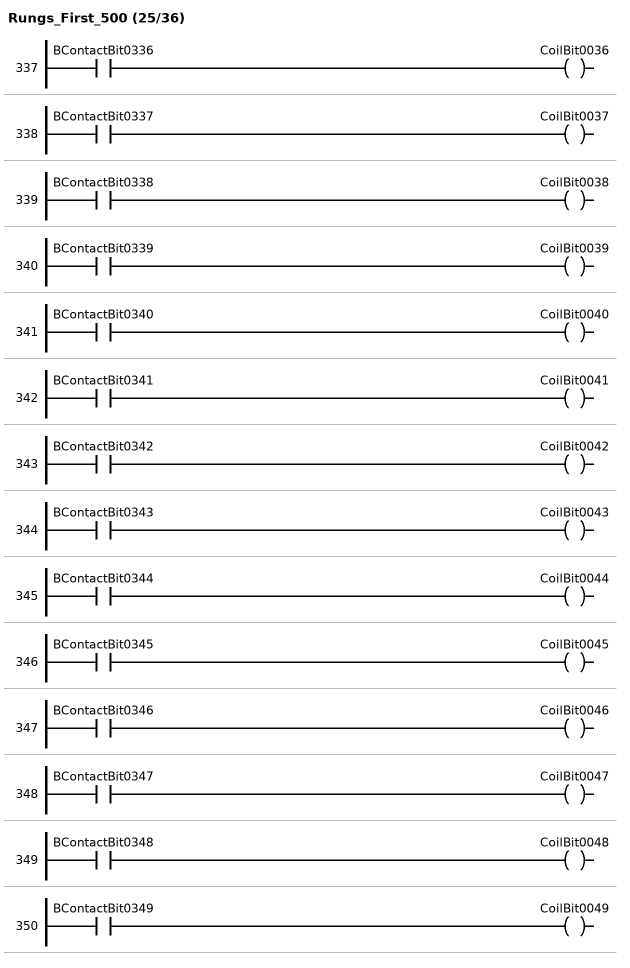
// NETWORK 337
CoilBit0036 := BContactBit0336;

// NETWORK 338
CoilBit0037 := BContactBit0337;

// NETWORK 339
CoilBit0038 := BContactBit0338;

// NETWORK 340
CoilBit0039 := BContactBit0339;

// NETWORK 341
CoilBit0040 := BContactBit0340;

// NETWORK 342
CoilBit0041 := BContactBit0341;

// NETWORK 343
CoilBit0042 := BContactBit0342;

// NETWORK 344
CoilBit0043 := BContactBit0343;

// NETWORK 345
CoilBit0044 := BContactBit0344;

// NETWORK 346
CoilBit0045 := BContactBit0345;

// NETWORK 347
CoilBit0046 := BContactBit0346;

// NETWORK 348
CoilBit0047 := BContactBit0347;

// NETWORK 349
CoilBit0048 := BContactBit0348;

// NETWORK 350
CoilBit0049 := BContactBit0349;

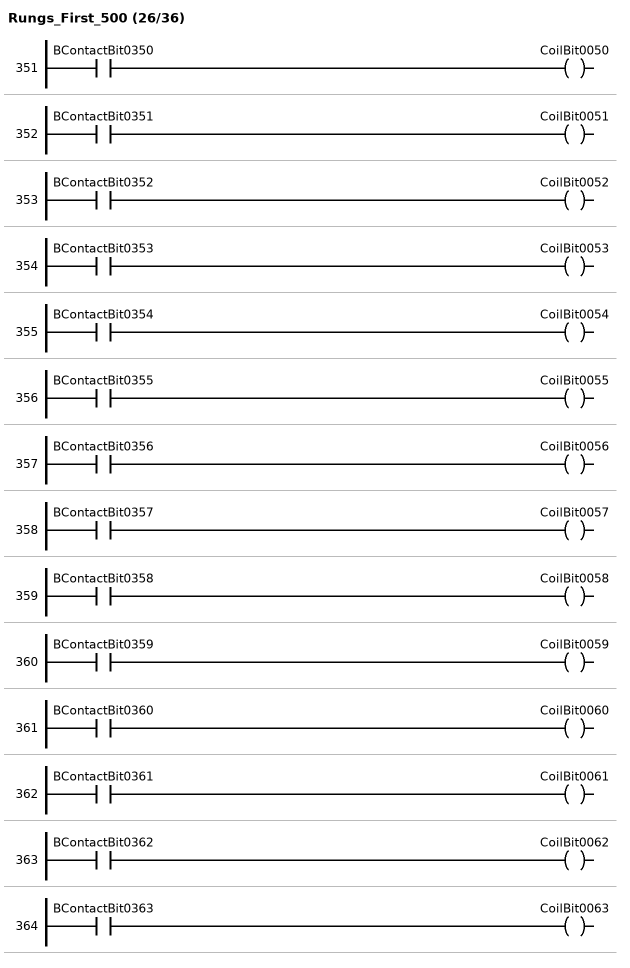
// NETWORK 351
CoilBit0050 := BContactBit0350;

// NETWORK 352
CoilBit0051 := BContactBit0351;

// NETWORK 353
CoilBit0052 := BContactBit0352;

// NETWORK 354
CoilBit0053 := BContactBit0353;

// NETWORK 355
CoilBit0054 := BContactBit0354;

// NETWORK 356
CoilBit0055 := BContactBit0355;

// NETWORK 357
CoilBit0056 := BContactBit0356;

// NETWORK 358
CoilBit0057 := BContactBit0357;

// NETWORK 359
CoilBit0058 := BContactBit0358;

// NETWORK 360
CoilBit0059 := BContactBit0359;

// NETWORK 361
CoilBit0060 := BContactBit0360;

// NETWORK 362
CoilBit0061 := BContactBit0361;

// NETWORK 363
CoilBit0062 := BContactBit0362;

// NETWORK 364
CoilBit0063 := BContactBit0363;

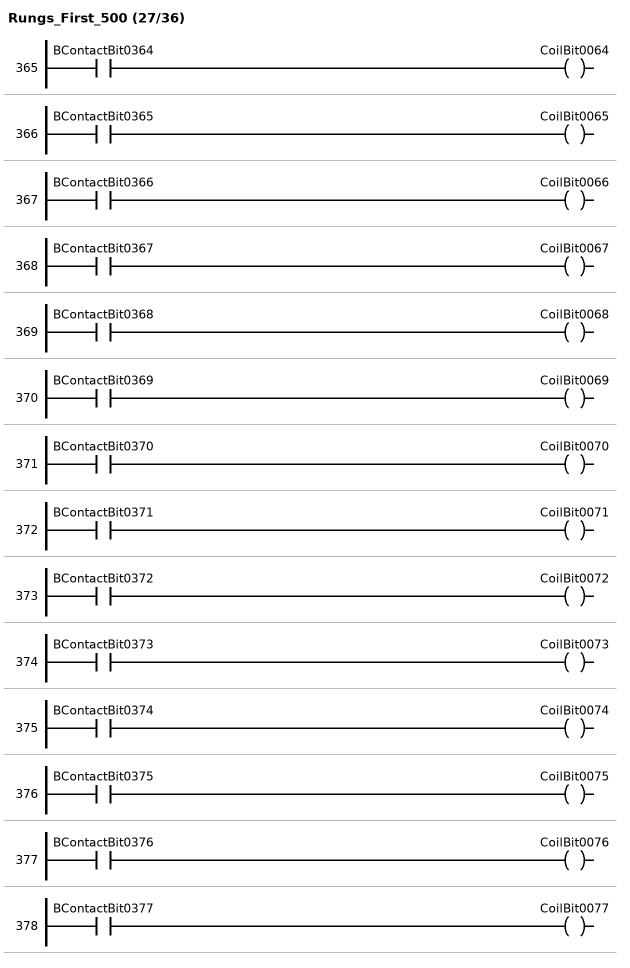
// NETWORK 365
CoilBit0064 := BContactBit0364;

// NETWORK 366
CoilBit0065 := BContactBit0365;

// NETWORK 367
CoilBit0066 := BContactBit0366;

// NETWORK 368
CoilBit0067 := BContactBit0367;

// NETWORK 369
CoilBit0068 := BContactBit0368;

// NETWORK 370
CoilBit0069 := BContactBit0369;

// NETWORK 371
CoilBit0070 := BContactBit0370;

// NETWORK 372
CoilBit0071 := BContactBit0371;

// NETWORK 373
CoilBit0072 := BContactBit0372;

// NETWORK 374
CoilBit0073 := BContactBit0373;

// NETWORK 375
CoilBit0074 := BContactBit0374;

// NETWORK 376
CoilBit0075 := BContactBit0375;

// NETWORK 377
CoilBit0076 := BContactBit0376;

// NETWORK 378
CoilBit0077 := BContactBit0377;

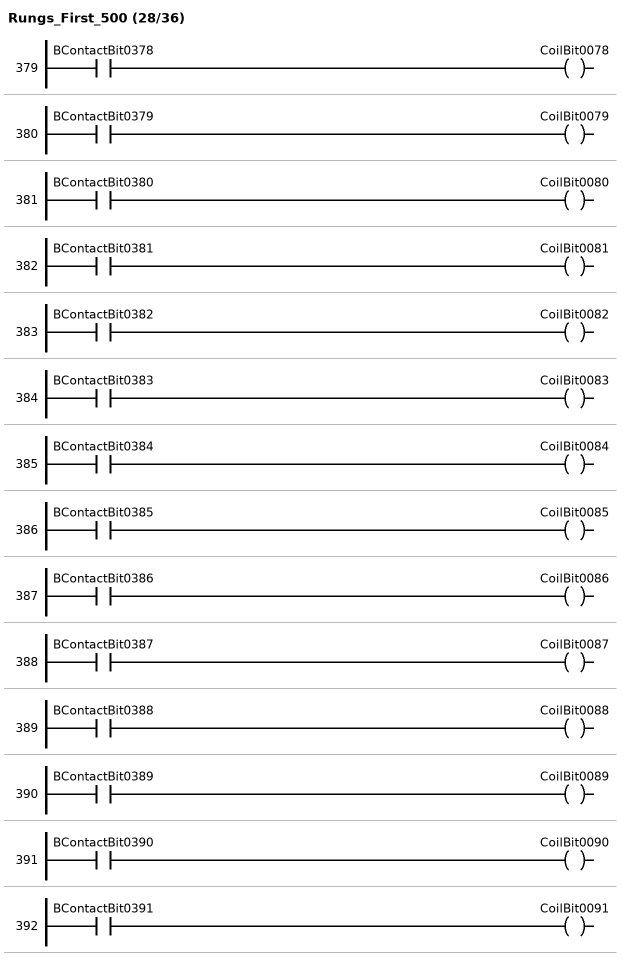
// NETWORK 379
CoilBit0078 := BContactBit0378;

// NETWORK 380
CoilBit0079 := BContactBit0379;

// NETWORK 381
CoilBit0080 := BContactBit0380;

// NETWORK 382
CoilBit0081 := BContactBit0381;

// NETWORK 383
CoilBit0082 := BContactBit0382;

// NETWORK 384
CoilBit0083 := BContactBit0383;

// NETWORK 385
CoilBit0084 := BContactBit0384;

// NETWORK 386
CoilBit0085 := BContactBit0385;

// NETWORK 387
CoilBit0086 := BContactBit0386;

// NETWORK 388
CoilBit0087 := BContactBit0387;

// NETWORK 389
CoilBit0088 := BContactBit0388;

// NETWORK 390
CoilBit0089 := BContactBit0389;

// NETWORK 391
CoilBit0090 := BContactBit0390;

// NETWORK 392
CoilBit0091 := BContactBit0391;

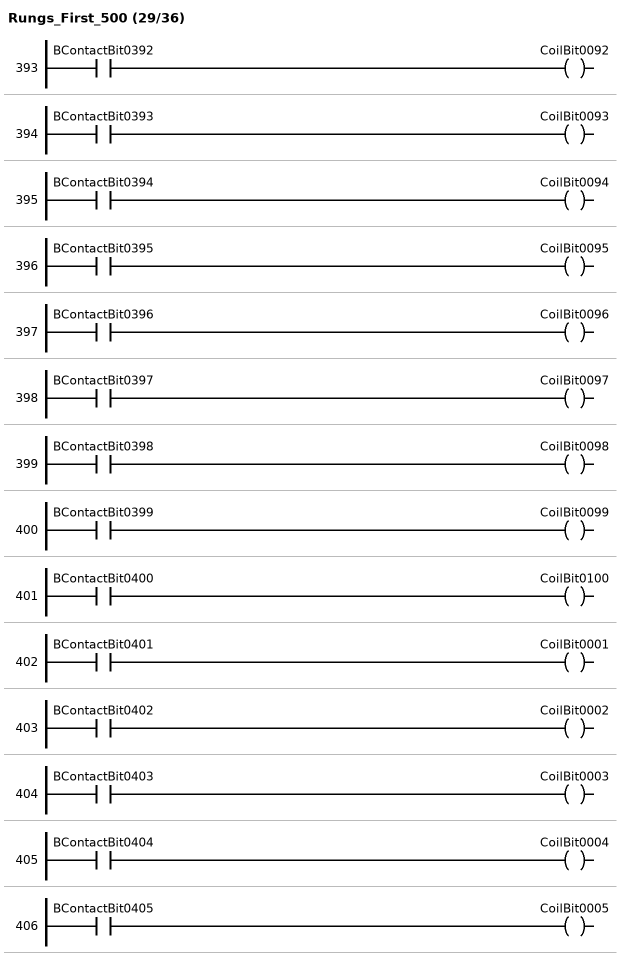
// NETWORK 393
CoilBit0092 := BContactBit0392;

// NETWORK 394
CoilBit0093 := BContactBit0393;

// NETWORK 395
CoilBit0094 := BContactBit0394;

// NETWORK 396
CoilBit0095 := BContactBit0395;

// NETWORK 397
CoilBit0096 := BContactBit0396;

// NETWORK 398
CoilBit0097 := BContactBit0397;

// NETWORK 399
CoilBit0098 := BContactBit0398;

// NETWORK 400
CoilBit0099 := BContactBit0399;

// NETWORK 401
CoilBit0100 := BContactBit0400;

// NETWORK 402
CoilBit0001 := BContactBit0401;

// NETWORK 403
CoilBit0002 := BContactBit0402;

// NETWORK 404
CoilBit0003 := BContactBit0403;

// NETWORK 405
CoilBit0004 := BContactBit0404;

// NETWORK 406
CoilBit0005 := BContactBit0405;

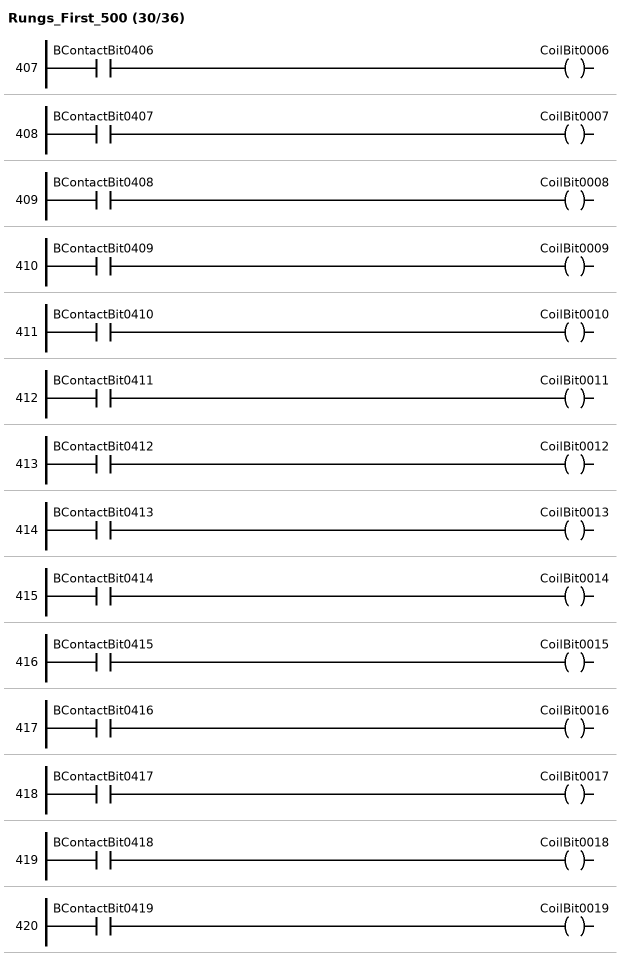
// NETWORK 407
CoilBit0006 := BContactBit0406;

// NETWORK 408
CoilBit0007 := BContactBit0407;

// NETWORK 409
CoilBit0008 := BContactBit0408;

// NETWORK 410
CoilBit0009 := BContactBit0409;

// NETWORK 411
CoilBit0010 := BContactBit0410;

// NETWORK 412
CoilBit0011 := BContactBit0411;

// NETWORK 413
CoilBit0012 := BContactBit0412;

// NETWORK 414
CoilBit0013 := BContactBit0413;

// NETWORK 415
CoilBit0014 := BContactBit0414;

// NETWORK 416
CoilBit0015 := BContactBit0415;

// NETWORK 417
CoilBit0016 := BContactBit0416;

// NETWORK 418
CoilBit0017 := BContactBit0417;

// NETWORK 419
CoilBit0018 := BContactBit0418;

// NETWORK 420
CoilBit0019 := BContactBit0419;

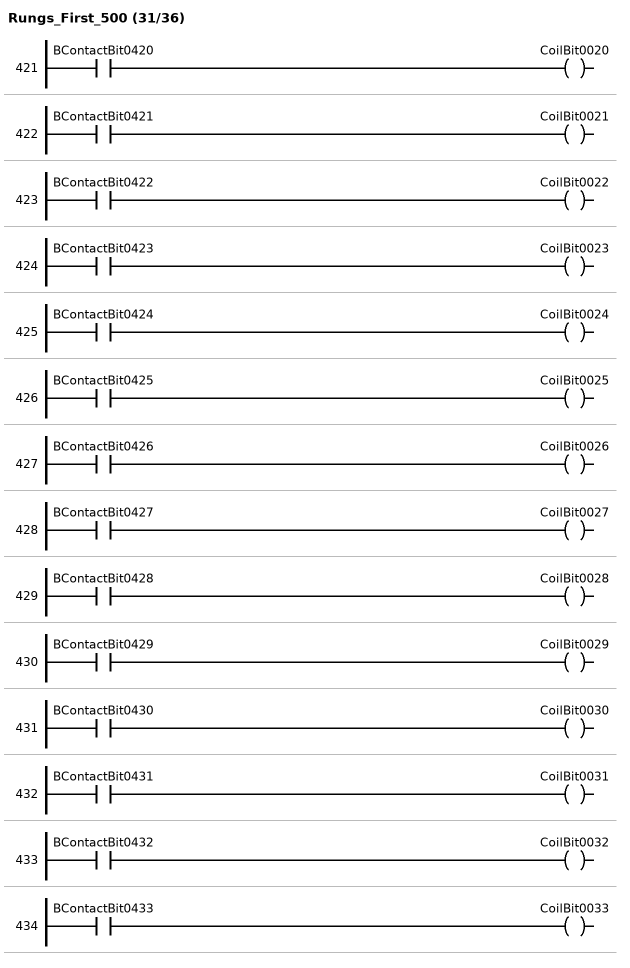
// NETWORK 421
CoilBit0020 := BContactBit0420;

// NETWORK 422
CoilBit0021 := BContactBit0421;

// NETWORK 423
CoilBit0022 := BContactBit0422;

// NETWORK 424
CoilBit0023 := BContactBit0423;

// NETWORK 425
CoilBit0024 := BContactBit0424;

// NETWORK 426
CoilBit0025 := BContactBit0425;

// NETWORK 427
CoilBit0026 := BContactBit0426;

// NETWORK 428
CoilBit0027 := BContactBit0427;

// NETWORK 429
CoilBit0028 := BContactBit0428;

// NETWORK 430
CoilBit0029 := BContactBit0429;

// NETWORK 431
CoilBit0030 := BContactBit0430;

// NETWORK 432
CoilBit0031 := BContactBit0431;

// NETWORK 433
CoilBit0032 := BContactBit0432;

// NETWORK 434
CoilBit0033 := BContactBit0433;

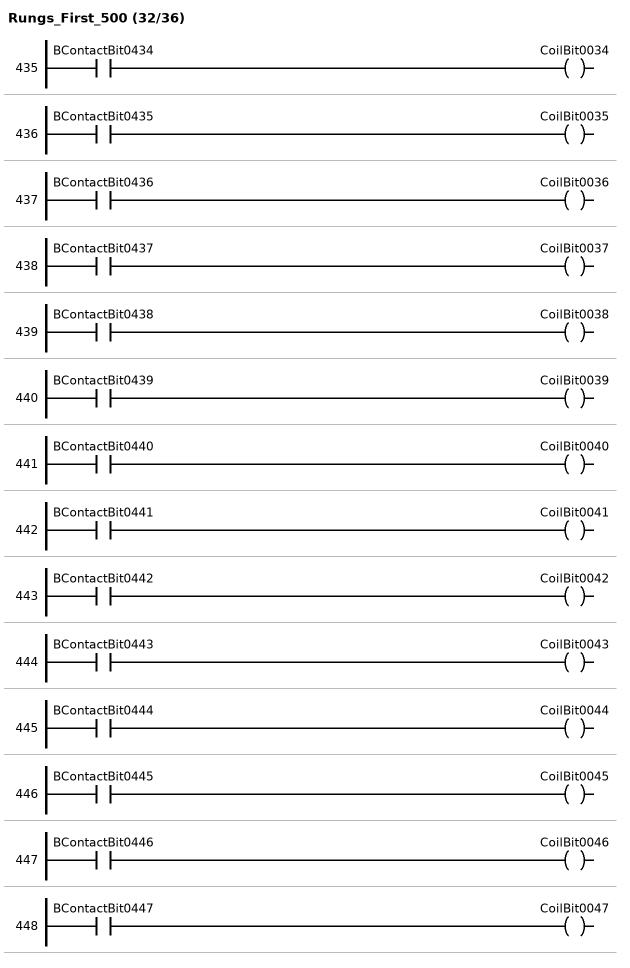
// NETWORK 435
CoilBit0034 := BContactBit0434;

// NETWORK 436
CoilBit0035 := BContactBit0435;

// NETWORK 437
CoilBit0036 := BContactBit0436;

// NETWORK 438
CoilBit0037 := BContactBit0437;

// NETWORK 439
CoilBit0038 := BContactBit0438;

// NETWORK 440
CoilBit0039 := BContactBit0439;

// NETWORK 441
CoilBit0040 := BContactBit0440;

// NETWORK 442
CoilBit0041 := BContactBit0441;

// NETWORK 443
CoilBit0042 := BContactBit0442;

// NETWORK 444
CoilBit0043 := BContactBit0443;

// NETWORK 445
CoilBit0044 := BContactBit0444;

// NETWORK 446
CoilBit0045 := BContactBit0445;

// NETWORK 447
CoilBit0046 := BContactBit0446;

// NETWORK 448
CoilBit0047 := BContactBit0447;

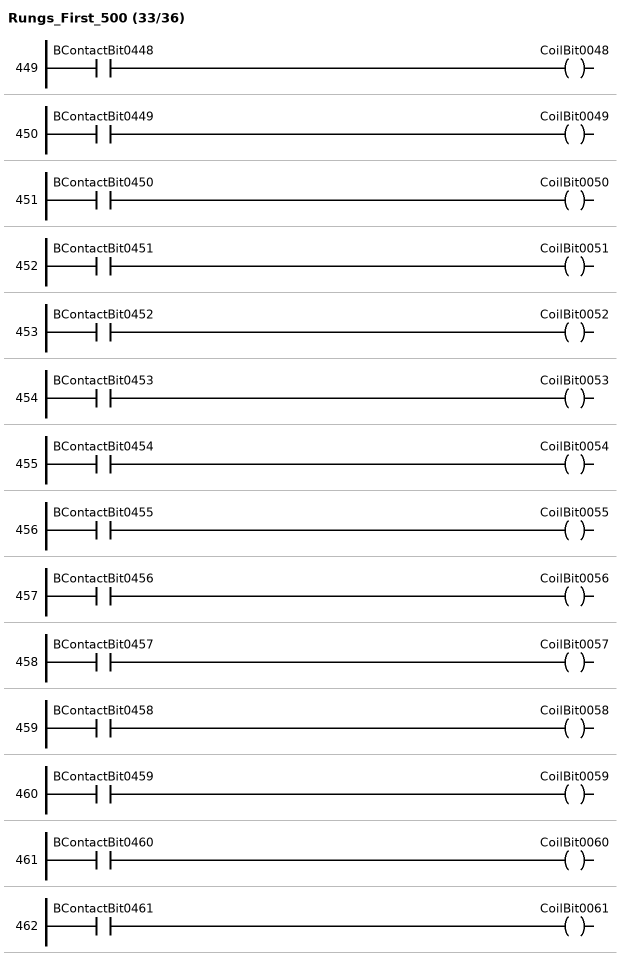
// NETWORK 449
CoilBit0048 := BContactBit0448;

// NETWORK 450
CoilBit0049 := BContactBit0449;

// NETWORK 451
CoilBit0050 := BContactBit0450;

// NETWORK 452
CoilBit0051 := BContactBit0451;

// NETWORK 453
CoilBit0052 := BContactBit0452;

// NETWORK 454
CoilBit0053 := BContactBit0453;

// NETWORK 455
CoilBit0054 := BContactBit0454;

// NETWORK 456
CoilBit0055 := BContactBit0455;

// NETWORK 457
CoilBit0056 := BContactBit0456;

// NETWORK 458
CoilBit0057 := BContactBit0457;

// NETWORK 459
CoilBit0058 := BContactBit0458;

// NETWORK 460
CoilBit0059 := BContactBit0459;

// NETWORK 461
CoilBit0060 := BContactBit0460;

// NETWORK 462
CoilBit0061 := BContactBit0461;

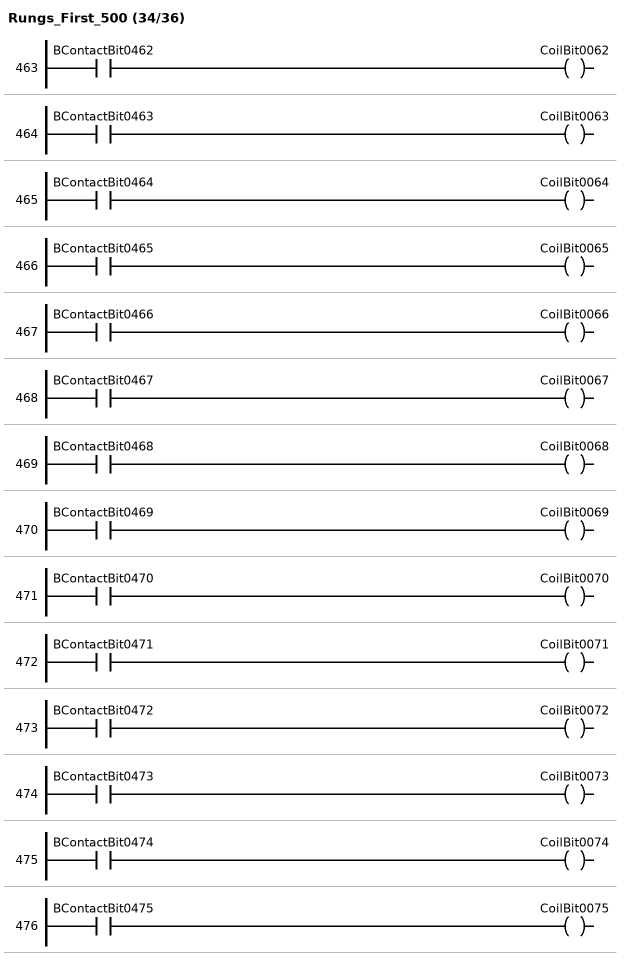
// NETWORK 463
CoilBit0062 := BContactBit0462;

// NETWORK 464
CoilBit0063 := BContactBit0463;

// NETWORK 465
CoilBit0064 := BContactBit0464;

// NETWORK 466
CoilBit0065 := BContactBit0465;

// NETWORK 467
CoilBit0066 := BContactBit0466;

// NETWORK 468
CoilBit0067 := BContactBit0467;

// NETWORK 469
CoilBit0068 := BContactBit0468;

// NETWORK 470
CoilBit0069 := BContactBit0469;

// NETWORK 471
CoilBit0070 := BContactBit0470;

// NETWORK 472
CoilBit0071 := BContactBit0471;

// NETWORK 473
CoilBit0072 := BContactBit0472;

// NETWORK 474
CoilBit0073 := BContactBit0473;

// NETWORK 475
CoilBit0074 := BContactBit0474;

// NETWORK 476
CoilBit0075 := BContactBit0475;

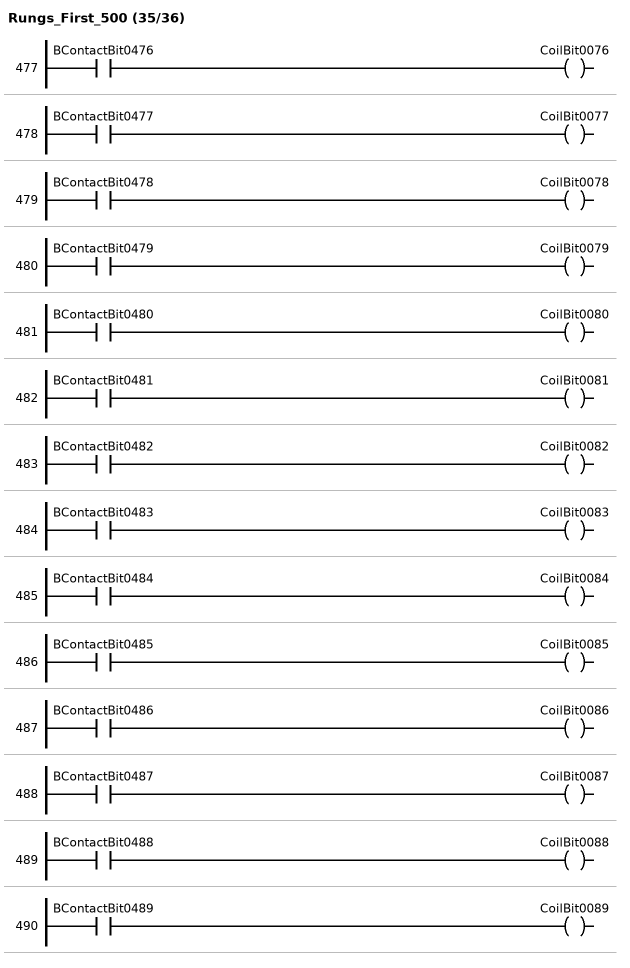
// NETWORK 477
CoilBit0076 := BContactBit0476;

// NETWORK 478
CoilBit0077 := BContactBit0477;

// NETWORK 479
CoilBit0078 := BContactBit0478;

// NETWORK 480
CoilBit0079 := BContactBit0479;

// NETWORK 481
CoilBit0080 := BContactBit0480;

// NETWORK 482
CoilBit0081 := BContactBit0481;

// NETWORK 483
CoilBit0082 := BContactBit0482;

// NETWORK 484
CoilBit0083 := BContactBit0483;

// NETWORK 485
CoilBit0084 := BContactBit0484;

// NETWORK 486
CoilBit0085 := BContactBit0485;

// NETWORK 487
CoilBit0086 := BContactBit0486;

// NETWORK 488
CoilBit0087 := BContactBit0487;

// NETWORK 489
CoilBit0088 := BContactBit0488;

// NETWORK 490
CoilBit0089 := BContactBit0489;

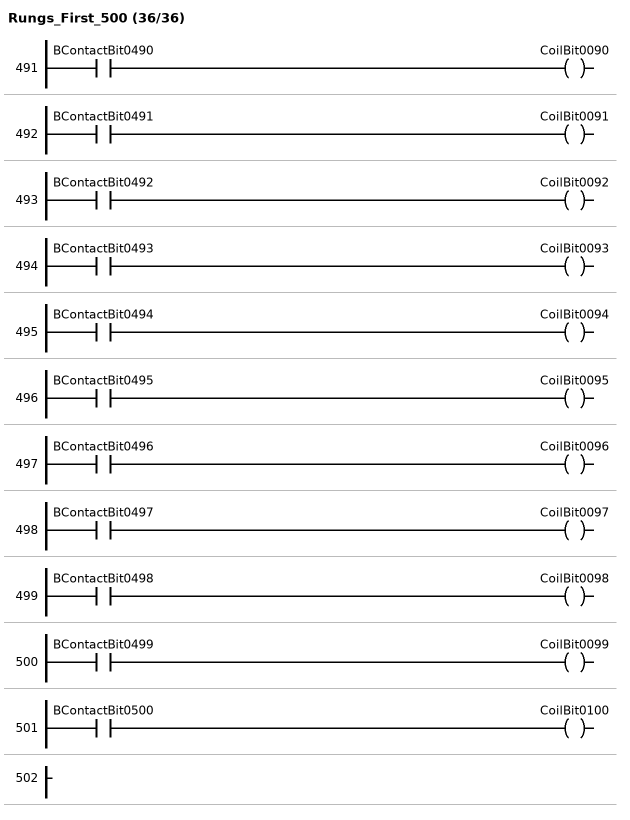
// NETWORK 491
CoilBit0090 := BContactBit0490;

// NETWORK 492
CoilBit0091 := BContactBit0491;

// NETWORK 493
CoilBit0092 := BContactBit0492;

// NETWORK 494
CoilBit0093 := BContactBit0493;

// NETWORK 495
CoilBit0094 := BContactBit0494;

// NETWORK 496
CoilBit0095 := BContactBit0495;

// NETWORK 497
CoilBit0096 := BContactBit0496;

// NETWORK 498
CoilBit0097 := BContactBit0497;

// NETWORK 499
CoilBit0098 := BContactBit0498;

// NETWORK 500
CoilBit0099 := BContactBit0499;

// NETWORK 501
CoilBit0100 := BContactBit0500;

// NETWORK 502

END_PROGRAM

// Rungs_Second_500
PROGRAM Rungs_Second_500
VAR

ContactBit0000	:BOOL;
ContactBit0001	:BOOL;
ContactBit0002	:BOOL;
ContactBit0003	:BOOL;
ContactBit0004	:BOOL;
ContactBit0005	:BOOL;
ContactBit0006	:BOOL;
ContactBit0007	:BOOL;
ContactBit0008	:BOOL;
ContactBit0009	:BOOL;
ContactBit0010	:BOOL;
ContactBit0011	:BOOL;
ContactBit0012	:BOOL;
ContactBit0013	:BOOL;
ContactBit0014	:BOOL;
ContactBit0015	:BOOL;
ContactBit0016	:BOOL;
ContactBit0017	:BOOL;
ContactBit0018	:BOOL;
ContactBit0019	:BOOL;
ContactBit0020	:BOOL;
ContactBit0021	:BOOL;
ContactBit0022	:BOOL;
ContactBit0023	:BOOL;
ContactBit0024	:BOOL;
ContactBit0025	:BOOL;
ContactBit0026	:BOOL;
ContactBit0027	:BOOL;
ContactBit0028	:BOOL;
ContactBit0029	:BOOL;
ContactBit0030	:BOOL;
ContactBit0031	:BOOL;
ContactBit0032	:BOOL;
ContactBit0033	:BOOL;
ContactBit0034	:BOOL;
ContactBit0035	:BOOL;
ContactBit0036	:BOOL;
ContactBit0037	:BOOL;
ContactBit0038	:BOOL;
ContactBit0039	:BOOL;
ContactBit0040	:BOOL;
ContactBit0041	:BOOL;
ContactBit0042	:BOOL;
ContactBit0043	:BOOL;
ContactBit0044	:BOOL;
ContactBit0045	:BOOL;
ContactBit0046	:BOOL;
ContactBit0047	:BOOL;
ContactBit0048	:BOOL;
ContactBit0049	:BOOL;
ContactBit0050	:BOOL;
ContactBit0051	:BOOL;
ContactBit0052	:BOOL;
ContactBit0053	:BOOL;
ContactBit0054	:BOOL;
ContactBit0055	:BOOL;
ContactBit0056	:BOOL;
ContactBit0057	:BOOL;
ContactBit0058	:BOOL;
ContactBit0059	:BOOL;
ContactBit0060	:BOOL;
ContactBit0061	:BOOL;
ContactBit0062	:BOOL;
ContactBit0063	:BOOL;
ContactBit0064	:BOOL;
ContactBit0065	:BOOL;
ContactBit0066	:BOOL;
ContactBit0067	:BOOL;
ContactBit0068	:BOOL;
ContactBit0069	:BOOL;
ContactBit0070	:BOOL;
ContactBit0071	:BOOL;
ContactBit0072	:BOOL;
ContactBit0073	:BOOL;
ContactBit0074	:BOOL;
ContactBit0075	:BOOL;
ContactBit0076	:BOOL;
ContactBit0077	:BOOL;
ContactBit0078	:BOOL;
ContactBit0079	:BOOL;
ContactBit0080	:BOOL;
ContactBit0081	:BOOL;
ContactBit0082	:BOOL;
ContactBit0083	:BOOL;
ContactBit0084	:BOOL;
ContactBit0085	:BOOL;
ContactBit0086	:BOOL;
ContactBit0087	:BOOL;
ContactBit0088	:BOOL;
ContactBit0089	:BOOL;
ContactBit0090	:BOOL;
ContactBit0091	:BOOL;
ContactBit0092	:BOOL;
ContactBit0093	:BOOL;
ContactBit0094	:BOOL;
ContactBit0095	:BOOL;
ContactBit0096	:BOOL;
ContactBit0097	:BOOL;
ContactBit0098	:BOOL;
ContactBit0099	:BOOL;
ContactBit0100	:BOOL;
ContactBit0101	:BOOL;
ContactBit0102	:BOOL;
ContactBit0103	:BOOL;
ContactBit0104	:BOOL;
ContactBit0105	:BOOL;
ContactBit0106	:BOOL;
ContactBit0107	:BOOL;
ContactBit0108	:BOOL;
ContactBit0109	:BOOL;
ContactBit0110	:BOOL;
ContactBit0111	:BOOL;
ContactBit0112	:BOOL;
ContactBit0113	:BOOL;
ContactBit0114	:BOOL;
ContactBit0115	:BOOL;
ContactBit0116	:BOOL;
ContactBit0117	:BOOL;
ContactBit0118	:BOOL;
ContactBit0119	:BOOL;
ContactBit0120	:BOOL;
ContactBit0121	:BOOL;
ContactBit0122	:BOOL;
ContactBit0123	:BOOL;
ContactBit0124	:BOOL;
ContactBit0125	:BOOL;
ContactBit0126	:BOOL;
ContactBit0127	:BOOL;
ContactBit0128	:BOOL;
ContactBit0129	:BOOL;
ContactBit0130	:BOOL;
ContactBit0131	:BOOL;
ContactBit0132	:BOOL;
ContactBit0133	:BOOL;
ContactBit0134	:BOOL;
ContactBit0135	:BOOL;
ContactBit0136	:BOOL;
ContactBit0137	:BOOL;
ContactBit0138	:BOOL;
ContactBit0139	:BOOL;
ContactBit0140	:BOOL;
ContactBit0141	:BOOL;
ContactBit0142	:BOOL;
ContactBit0143	:BOOL;
ContactBit0144	:BOOL;
ContactBit0145	:BOOL;
ContactBit0146	:BOOL;
ContactBit0147	:BOOL;
ContactBit0148	:BOOL;
ContactBit0149	:BOOL;
ContactBit0150	:BOOL;
ContactBit0151	:BOOL;
ContactBit0152	:BOOL;
ContactBit0153	:BOOL;
ContactBit0154	:BOOL;
ContactBit0155	:BOOL;
ContactBit0156	:BOOL;
ContactBit0157	:BOOL;
ContactBit0158	:BOOL;
ContactBit0159	:BOOL;
ContactBit0160	:BOOL;
ContactBit0161	:BOOL;
ContactBit0162	:BOOL;
ContactBit0163	:BOOL;
ContactBit0164	:BOOL;
ContactBit0165	:BOOL;
ContactBit0166	:BOOL;
ContactBit0167	:BOOL;
ContactBit0168	:BOOL;
ContactBit0169	:BOOL;
ContactBit0170	:BOOL;
ContactBit0171	:BOOL;
ContactBit0172	:BOOL;
ContactBit0173	:BOOL;
ContactBit0174	:BOOL;
ContactBit0175	:BOOL;
ContactBit0176	:BOOL;
ContactBit0177	:BOOL;
ContactBit0178	:BOOL;
ContactBit0179	:BOOL;
ContactBit0180	:BOOL;
ContactBit0181	:BOOL;
ContactBit0182	:BOOL;
ContactBit0183	:BOOL;
ContactBit0184	:BOOL;
ContactBit0185	:BOOL;
ContactBit0186	:BOOL;
ContactBit0187	:BOOL;
ContactBit0188	:BOOL;
ContactBit0189	:BOOL;
ContactBit0190	:BOOL;
ContactBit0191	:BOOL;
ContactBit0192	:BOOL;
ContactBit0193	:BOOL;
ContactBit0194	:BOOL;
ContactBit0195	:BOOL;
ContactBit0196	:BOOL;
ContactBit0197	:BOOL;
ContactBit0198	:BOOL;
ContactBit0199	:BOOL;
ContactBit0200	:BOOL;
ContactBit0201	:BOOL;
ContactBit0202	:BOOL;
ContactBit0203	:BOOL;
ContactBit0204	:BOOL;
ContactBit0205	:BOOL;
ContactBit0206	:BOOL;
ContactBit0207	:BOOL;
ContactBit0208	:BOOL;
ContactBit0209	:BOOL;
ContactBit0210	:BOOL;
ContactBit0211	:BOOL;
ContactBit0212	:BOOL;
ContactBit0213	:BOOL;
ContactBit0214	:BOOL;
ContactBit0215	:BOOL;
ContactBit0216	:BOOL;
ContactBit0217	:BOOL;
ContactBit0218	:BOOL;
ContactBit0219	:BOOL;
ContactBit0220	:BOOL;
ContactBit0221	:BOOL;
ContactBit0222	:BOOL;
ContactBit0223	:BOOL;
ContactBit0224	:BOOL;
ContactBit0225	:BOOL;
ContactBit0226	:BOOL;
ContactBit0227	:BOOL;
ContactBit0228	:BOOL;
ContactBit0229	:BOOL;
ContactBit0230	:BOOL;
ContactBit0231	:BOOL;
ContactBit0232	:BOOL;
ContactBit0233	:BOOL;
ContactBit0234	:BOOL;
ContactBit0235	:BOOL;
ContactBit0236	:BOOL;
ContactBit0237	:BOOL;
ContactBit0238	:BOOL;
ContactBit0239	:BOOL;
ContactBit0240	:BOOL;
ContactBit0241	:BOOL;
ContactBit0242	:BOOL;
ContactBit0243	:BOOL;
ContactBit0244	:BOOL;
ContactBit0245	:BOOL;
ContactBit0246	:BOOL;
ContactBit0247	:BOOL;
ContactBit0248	:BOOL;
ContactBit0249	:BOOL;
ContactBit0250	:BOOL;
ContactBit0251	:BOOL;
ContactBit0252	:BOOL;
ContactBit0253	:BOOL;
ContactBit0254	:BOOL;
ContactBit0255	:BOOL;
ContactBit0256	:BOOL;
ContactBit0257	:BOOL;
ContactBit0258	:BOOL;
ContactBit0259	:BOOL;
ContactBit0260	:BOOL;
ContactBit0261	:BOOL;
ContactBit0262	:BOOL;
ContactBit0263	:BOOL;
ContactBit0264	:BOOL;
ContactBit0265	:BOOL;
ContactBit0266	:BOOL;
ContactBit0267	:BOOL;
ContactBit0268	:BOOL;
ContactBit0269	:BOOL;
ContactBit0270	:BOOL;
ContactBit0271	:BOOL;
ContactBit0272	:BOOL;
ContactBit0273	:BOOL;
ContactBit0274	:BOOL;
ContactBit0275	:BOOL;
ContactBit0276	:BOOL;
ContactBit0277	:BOOL;
ContactBit0278	:BOOL;
ContactBit0279	:BOOL;
ContactBit0280	:BOOL;
ContactBit0281	:BOOL;
ContactBit0282	:BOOL;
ContactBit0283	:BOOL;
ContactBit0284	:BOOL;
ContactBit0285	:BOOL;
ContactBit0286	:BOOL;
ContactBit0287	:BOOL;
ContactBit0288	:BOOL;
ContactBit0289	:BOOL;
ContactBit0290	:BOOL;
ContactBit0291	:BOOL;
ContactBit0292	:BOOL;
ContactBit0293	:BOOL;
ContactBit0294	:BOOL;
ContactBit0295	:BOOL;
ContactBit0296	:BOOL;
ContactBit0297	:BOOL;
ContactBit0298	:BOOL;
ContactBit0299	:BOOL;
ContactBit0300	:BOOL;
ContactBit0301	:BOOL;
ContactBit0302	:BOOL;
ContactBit0303	:BOOL;
ContactBit0304	:BOOL;
ContactBit0305	:BOOL;
ContactBit0306	:BOOL;
ContactBit0307	:BOOL;
ContactBit0308	:BOOL;
ContactBit0309	:BOOL;
ContactBit0310	:BOOL;
ContactBit0311	:BOOL;
ContactBit0312	:BOOL;
ContactBit0313	:BOOL;
ContactBit0314	:BOOL;
ContactBit0315	:BOOL;
ContactBit0316	:BOOL;
ContactBit0317	:BOOL;
ContactBit0318	:BOOL;
ContactBit0319	:BOOL;
ContactBit0320	:BOOL;
ContactBit0321	:BOOL;
ContactBit0322	:BOOL;
ContactBit0323	:BOOL;
ContactBit0324	:BOOL;
ContactBit0325	:BOOL;
ContactBit0326	:BOOL;
ContactBit0327	:BOOL;
ContactBit0328	:BOOL;
ContactBit0329	:BOOL;
ContactBit0330	:BOOL;
ContactBit0331	:BOOL;
ContactBit0332	:BOOL;
ContactBit0333	:BOOL;
ContactBit0334	:BOOL;
ContactBit0335	:BOOL;
ContactBit0336	:BOOL;
ContactBit0337	:BOOL;
ContactBit0338	:BOOL;
ContactBit0339	:BOOL;
ContactBit0340	:BOOL;
ContactBit0341	:BOOL;
ContactBit0342	:BOOL;
ContactBit0343	:BOOL;
ContactBit0344	:BOOL;
ContactBit0345	:BOOL;
ContactBit0346	:BOOL;
ContactBit0347	:BOOL;
ContactBit0348	:BOOL;
ContactBit0349	:BOOL;
ContactBit0350	:BOOL;
ContactBit0351	:BOOL;
ContactBit0352	:BOOL;
ContactBit0353	:BOOL;
ContactBit0354	:BOOL;
ContactBit0355	:BOOL;
ContactBit0356	:BOOL;
ContactBit0357	:BOOL;
ContactBit0358	:BOOL;
ContactBit0359	:BOOL;
ContactBit0360	:BOOL;
ContactBit0361	:BOOL;
ContactBit0362	:BOOL;
ContactBit0363	:BOOL;
ContactBit0364	:BOOL;
ContactBit0365	:BOOL;
ContactBit0366	:BOOL;
ContactBit0367	:BOOL;
ContactBit0368	:BOOL;
ContactBit0369	:BOOL;
ContactBit0370	:BOOL;
ContactBit0371	:BOOL;
ContactBit0372	:BOOL;
ContactBit0373	:BOOL;
ContactBit0374	:BOOL;
ContactBit0375	:BOOL;
ContactBit0376	:BOOL;
ContactBit0377	:BOOL;
ContactBit0378	:BOOL;
ContactBit0379	:BOOL;
ContactBit0380	:BOOL;
ContactBit0381	:BOOL;
ContactBit0382	:BOOL;
ContactBit0383	:BOOL;
ContactBit0384	:BOOL;
ContactBit0385	:BOOL;
ContactBit0386	:BOOL;
ContactBit0387	:BOOL;
ContactBit0388	:BOOL;
ContactBit0389	:BOOL;
ContactBit0390	:BOOL;
ContactBit0391	:BOOL;
ContactBit0392	:BOOL;
ContactBit0393	:BOOL;
ContactBit0394	:BOOL;
ContactBit0395	:BOOL;
ContactBit0396	:BOOL;
ContactBit0397	:BOOL;
ContactBit0398	:BOOL;
ContactBit0399	:BOOL;
ContactBit0400	:BOOL;
ContactBit0401	:BOOL;
ContactBit0402	:BOOL;
ContactBit0403	:BOOL;
ContactBit0404	:BOOL;
ContactBit0405	:BOOL;
ContactBit0406	:BOOL;
ContactBit0407	:BOOL;
ContactBit0408	:BOOL;
ContactBit0409	:BOOL;
ContactBit0410	:BOOL;
ContactBit0411	:BOOL;
ContactBit0412	:BOOL;
ContactBit0413	:BOOL;
ContactBit0414	:BOOL;
ContactBit0415	:BOOL;
ContactBit0416	:BOOL;
ContactBit0417	:BOOL;
ContactBit0418	:BOOL;
ContactBit0419	:BOOL;
ContactBit0420	:BOOL;
ContactBit0421	:BOOL;
ContactBit0422	:BOOL;
ContactBit0423	:BOOL;
ContactBit0424	:BOOL;
ContactBit0425	:BOOL;
ContactBit0426	:BOOL;
ContactBit0427	:BOOL;
ContactBit0428	:BOOL;
ContactBit0429	:BOOL;
ContactBit0430	:BOOL;
ContactBit0431	:BOOL;
ContactBit0432	:BOOL;
ContactBit0433	:BOOL;
ContactBit0434	:BOOL;
ContactBit0435	:BOOL;
ContactBit0436	:BOOL;
ContactBit0437	:BOOL;
ContactBit0438	:BOOL;
ContactBit0439	:BOOL;
ContactBit0440	:BOOL;
ContactBit0441	:BOOL;
ContactBit0442	:BOOL;
ContactBit0443	:BOOL;
ContactBit0444	:BOOL;
ContactBit0445	:BOOL;
ContactBit0446	:BOOL;
ContactBit0447	:BOOL;
ContactBit0448	:BOOL;
ContactBit0449	:BOOL;
ContactBit0450	:BOOL;
ContactBit0451	:BOOL;
ContactBit0452	:BOOL;
ContactBit0453	:BOOL;
ContactBit0454	:BOOL;
ContactBit0455	:BOOL;
ContactBit0456	:BOOL;
ContactBit0457	:BOOL;
ContactBit0458	:BOOL;
ContactBit0459	:BOOL;
ContactBit0460	:BOOL;
ContactBit0461	:BOOL;
ContactBit0462	:BOOL;
ContactBit0463	:BOOL;
ContactBit0464	:BOOL;
ContactBit0465	:BOOL;
ContactBit0466	:BOOL;
ContactBit0467	:BOOL;
ContactBit0468	:BOOL;
ContactBit0469	:BOOL;
ContactBit0470	:BOOL;
ContactBit0471	:BOOL;
ContactBit0472	:BOOL;
ContactBit0473	:BOOL;
ContactBit0474	:BOOL;
ContactBit0475	:BOOL;
ContactBit0476	:BOOL;
ContactBit0477	:BOOL;
ContactBit0478	:BOOL;
ContactBit0479	:BOOL;
ContactBit0480	:BOOL;
ContactBit0481	:BOOL;
ContactBit0482	:BOOL;
ContactBit0483	:BOOL;
ContactBit0484	:BOOL;
ContactBit0485	:BOOL;
ContactBit0486	:BOOL;
ContactBit0487	:BOOL;
ContactBit0488	:BOOL;
ContactBit0489	:BOOL;
ContactBit0490	:BOOL;
ContactBit0491	:BOOL;
ContactBit0492	:BOOL;
ContactBit0493	:BOOL;
ContactBit0494	:BOOL;
ContactBit0495	:BOOL;
ContactBit0496	:BOOL;
ContactBit0497	:BOOL;
ContactBit0498	:BOOL;
ContactBit0499	:BOOL;
ContactBit0500	:BOOL;



CoilBit0000	:BOOL;
CoilBit0001	:BOOL;
CoilBit0002	:BOOL;
CoilBit0003	:BOOL;
CoilBit0004	:BOOL;
CoilBit0005	:BOOL;
CoilBit0006	:BOOL;
CoilBit0007	:BOOL;
CoilBit0008	:BOOL;
CoilBit0009	:BOOL;
CoilBit0010	:BOOL;
CoilBit0011	:BOOL;
CoilBit0012	:BOOL;
CoilBit0013	:BOOL;
CoilBit0014	:BOOL;
CoilBit0015	:BOOL;
CoilBit0016	:BOOL;
CoilBit0017	:BOOL;
CoilBit0018	:BOOL;
CoilBit0019	:BOOL;
CoilBit0020	:BOOL;
CoilBit0021	:BOOL;
CoilBit0022	:BOOL;
CoilBit0023	:BOOL;
CoilBit0024	:BOOL;
CoilBit0025	:BOOL;
CoilBit0026	:BOOL;
CoilBit0027	:BOOL;
CoilBit0028	:BOOL;
CoilBit0029	:BOOL;
CoilBit0030	:BOOL;
CoilBit0031	:BOOL;
CoilBit0032	:BOOL;
CoilBit0033	:BOOL;
CoilBit0034	:BOOL;
CoilBit0035	:BOOL;
CoilBit0036	:BOOL;
CoilBit0037	:BOOL;
CoilBit0038	:BOOL;
CoilBit0039	:BOOL;
CoilBit0040	:BOOL;
CoilBit0041	:BOOL;
CoilBit0042	:BOOL;
CoilBit0043	:BOOL;
CoilBit0044	:BOOL;
CoilBit0045	:BOOL;
CoilBit0046	:BOOL;
CoilBit0047	:BOOL;
CoilBit0048	:BOOL;
CoilBit0049	:BOOL;
CoilBit0050	:BOOL;
CoilBit0051	:BOOL;
CoilBit0052	:BOOL;
CoilBit0053	:BOOL;
CoilBit0054	:BOOL;
CoilBit0055	:BOOL;
CoilBit0056	:BOOL;
CoilBit0057	:BOOL;
CoilBit0058	:BOOL;
CoilBit0059	:BOOL;
CoilBit0060	:BOOL;
CoilBit0061	:BOOL;
CoilBit0062	:BOOL;
CoilBit0063	:BOOL;
CoilBit0064	:BOOL;
CoilBit0065	:BOOL;
CoilBit0066	:BOOL;
CoilBit0067	:BOOL;
CoilBit0068	:BOOL;
CoilBit0069	:BOOL;
CoilBit0070	:BOOL;
CoilBit0071	:BOOL;
CoilBit0072	:BOOL;
CoilBit0073	:BOOL;
CoilBit0074	:BOOL;
CoilBit0075	:BOOL;
CoilBit0076	:BOOL;
CoilBit0077	:BOOL;
CoilBit0078	:BOOL;
CoilBit0079	:BOOL;
CoilBit0080	:BOOL;
CoilBit0081	:BOOL;
CoilBit0082	:BOOL;
CoilBit0083	:BOOL;
CoilBit0084	:BOOL;
CoilBit0085	:BOOL;
CoilBit0086	:BOOL;
CoilBit0087	:BOOL;
CoilBit0088	:BOOL;
CoilBit0089	:BOOL;
CoilBit0090	:BOOL;
CoilBit0091	:BOOL;
CoilBit0092	:BOOL;
CoilBit0093	:BOOL;
CoilBit0094	:BOOL;
CoilBit0095	:BOOL;
CoilBit0096	:BOOL;
CoilBit0097	:BOOL;
CoilBit0098	:BOOL;
CoilBit0099	:BOOL;
CoilBit0100	:BOOL;

END_VAR

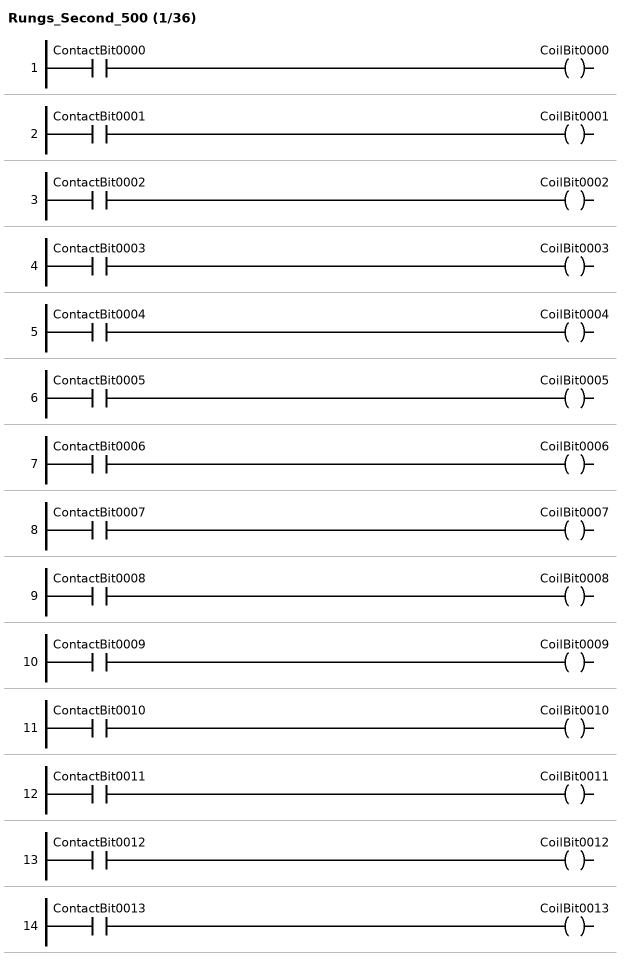
// NETWORK 1
CoilBit0000 := ContactBit0000;

// NETWORK 2
CoilBit0001 := ContactBit0001;

// NETWORK 3
CoilBit0002 := ContactBit0002;

// NETWORK 4
CoilBit0003 := ContactBit0003;

// NETWORK 5
CoilBit0004 := ContactBit0004;

// NETWORK 6
CoilBit0005 := ContactBit0005;

// NETWORK 7
CoilBit0006 := ContactBit0006;

// NETWORK 8
CoilBit0007 := ContactBit0007;

// NETWORK 9
CoilBit0008 := ContactBit0008;

// NETWORK 10
CoilBit0009 := ContactBit0009;

// NETWORK 11
CoilBit0010 := ContactBit0010;

// NETWORK 12
CoilBit0011 := ContactBit0011;

// NETWORK 13
CoilBit0012 := ContactBit0012;

// NETWORK 14
CoilBit0013 := ContactBit0013;

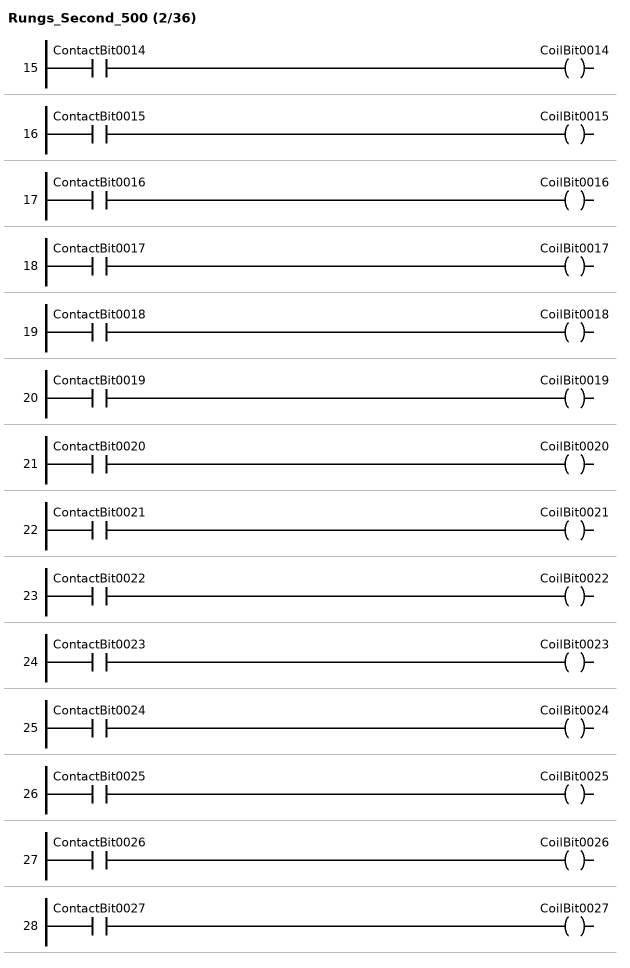
// NETWORK 15
CoilBit0014 := ContactBit0014;

// NETWORK 16
CoilBit0015 := ContactBit0015;

// NETWORK 17
CoilBit0016 := ContactBit0016;

// NETWORK 18
CoilBit0017 := ContactBit0017;

// NETWORK 19
CoilBit0018 := ContactBit0018;

// NETWORK 20
CoilBit0019 := ContactBit0019;

// NETWORK 21
CoilBit0020 := ContactBit0020;

// NETWORK 22
CoilBit0021 := ContactBit0021;

// NETWORK 23
CoilBit0022 := ContactBit0022;

// NETWORK 24
CoilBit0023 := ContactBit0023;

// NETWORK 25
CoilBit0024 := ContactBit0024;

// NETWORK 26
CoilBit0025 := ContactBit0025;

// NETWORK 27
CoilBit0026 := ContactBit0026;

// NETWORK 28
CoilBit0027 := ContactBit0027;

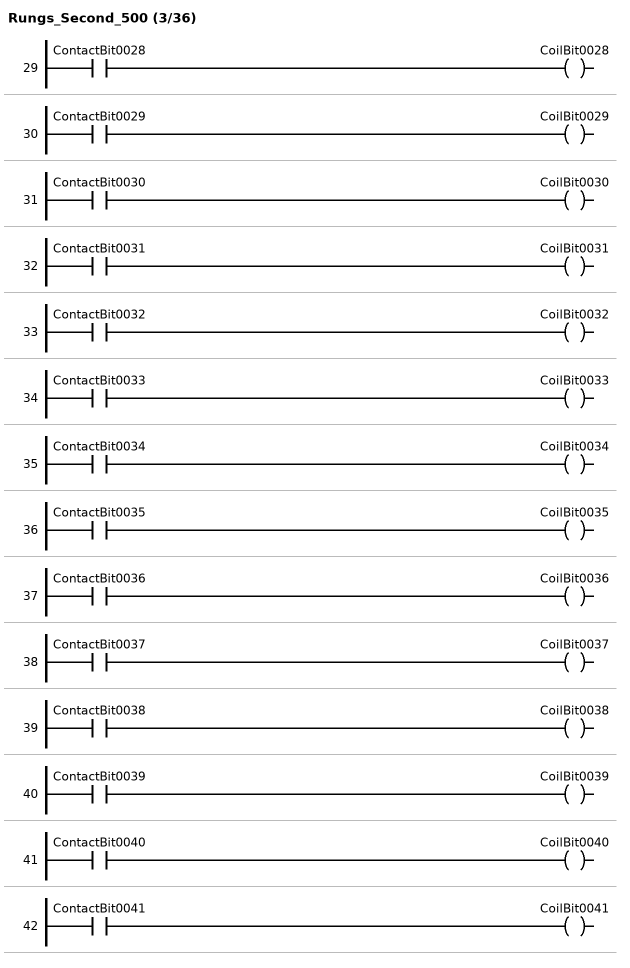
// NETWORK 29
CoilBit0028 := ContactBit0028;

// NETWORK 30
CoilBit0029 := ContactBit0029;

// NETWORK 31
CoilBit0030 := ContactBit0030;

// NETWORK 32
CoilBit0031 := ContactBit0031;

// NETWORK 33
CoilBit0032 := ContactBit0032;

// NETWORK 34
CoilBit0033 := ContactBit0033;

// NETWORK 35
CoilBit0034 := ContactBit0034;

// NETWORK 36
CoilBit0035 := ContactBit0035;

// NETWORK 37
CoilBit0036 := ContactBit0036;

// NETWORK 38
CoilBit0037 := ContactBit0037;

// NETWORK 39
CoilBit0038 := ContactBit0038;

// NETWORK 40
CoilBit0039 := ContactBit0039;

// NETWORK 41
CoilBit0040 := ContactBit0040;

// NETWORK 42
CoilBit0041 := ContactBit0041;

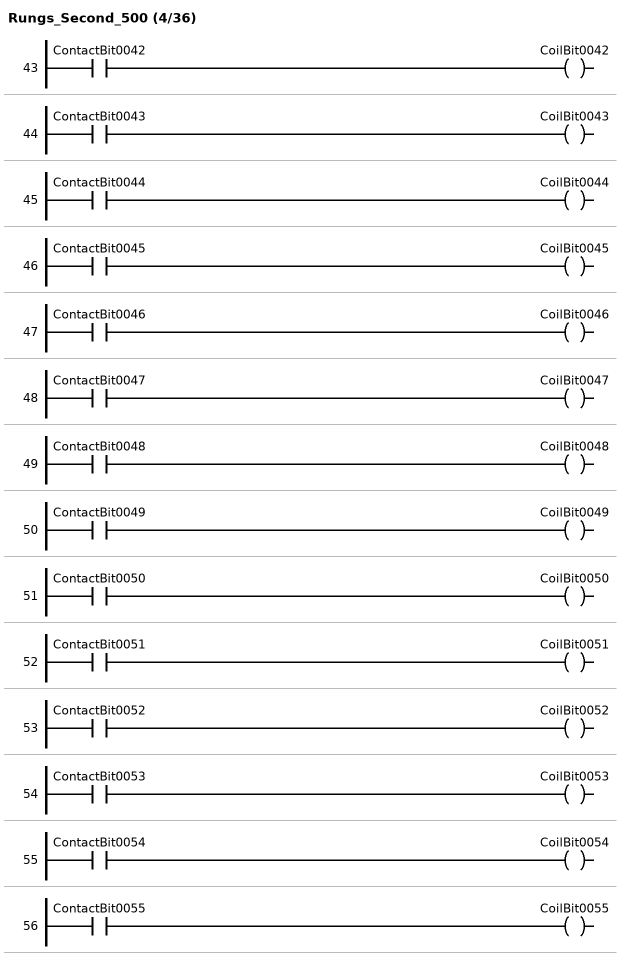
// NETWORK 43
CoilBit0042 := ContactBit0042;

// NETWORK 44
CoilBit0043 := ContactBit0043;

// NETWORK 45
CoilBit0044 := ContactBit0044;

// NETWORK 46
CoilBit0045 := ContactBit0045;

// NETWORK 47
CoilBit0046 := ContactBit0046;

// NETWORK 48
CoilBit0047 := ContactBit0047;

// NETWORK 49
CoilBit0048 := ContactBit0048;

// NETWORK 50
CoilBit0049 := ContactBit0049;

// NETWORK 51
CoilBit0050 := ContactBit0050;

// NETWORK 52
CoilBit0051 := ContactBit0051;

// NETWORK 53
CoilBit0052 := ContactBit0052;

// NETWORK 54
CoilBit0053 := ContactBit0053;

// NETWORK 55
CoilBit0054 := ContactBit0054;

// NETWORK 56
CoilBit0055 := ContactBit0055;

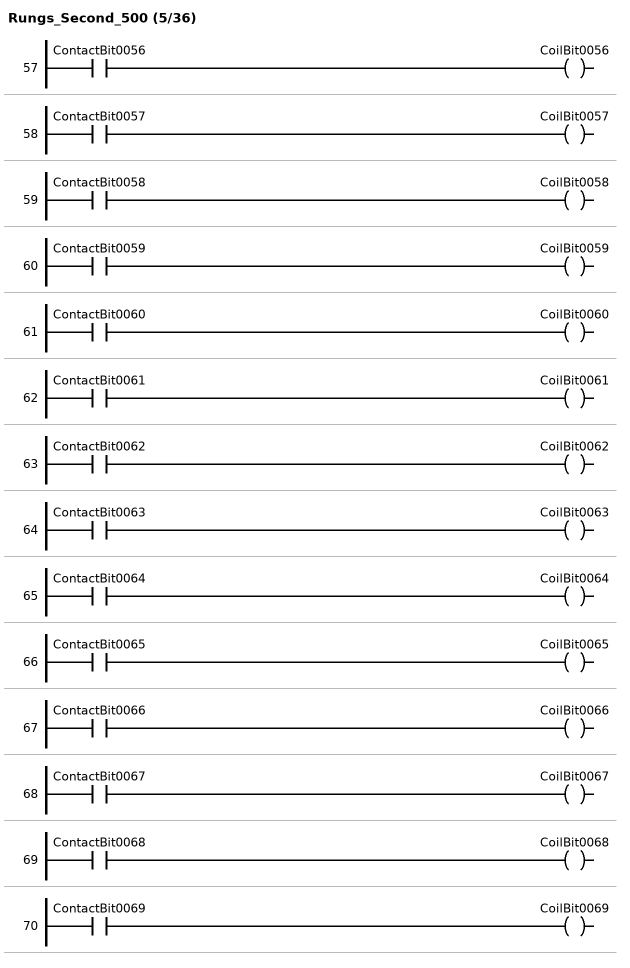
// NETWORK 57
CoilBit0056 := ContactBit0056;

// NETWORK 58
CoilBit0057 := ContactBit0057;

// NETWORK 59
CoilBit0058 := ContactBit0058;

// NETWORK 60
CoilBit0059 := ContactBit0059;

// NETWORK 61
CoilBit0060 := ContactBit0060;

// NETWORK 62
CoilBit0061 := ContactBit0061;

// NETWORK 63
CoilBit0062 := ContactBit0062;

// NETWORK 64
CoilBit0063 := ContactBit0063;

// NETWORK 65
CoilBit0064 := ContactBit0064;

// NETWORK 66
CoilBit0065 := ContactBit0065;

// NETWORK 67
CoilBit0066 := ContactBit0066;

// NETWORK 68
CoilBit0067 := ContactBit0067;

// NETWORK 69
CoilBit0068 := ContactBit0068;

// NETWORK 70
CoilBit0069 := ContactBit0069;

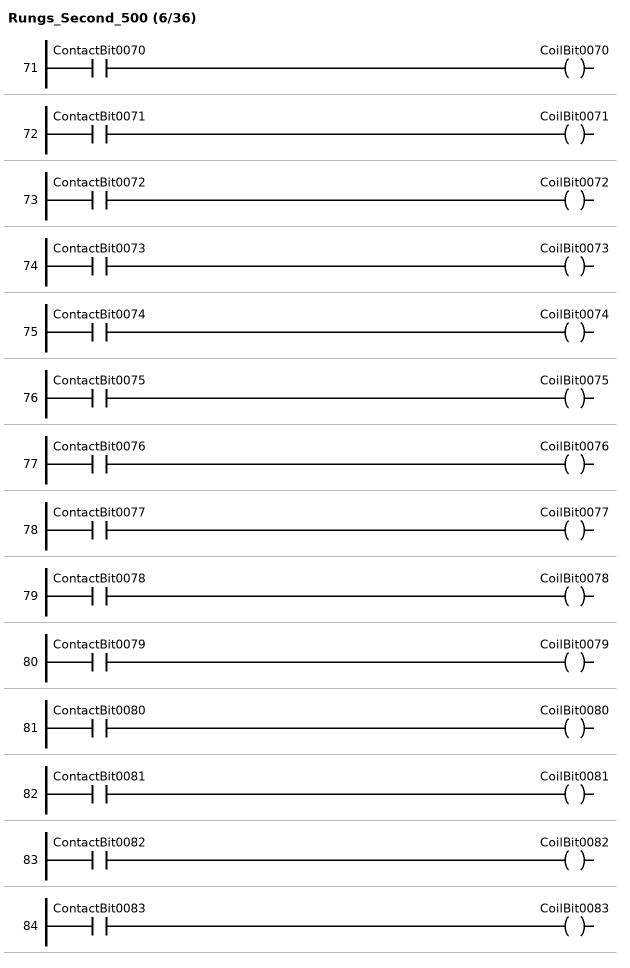
// NETWORK 71
CoilBit0070 := ContactBit0070;

// NETWORK 72
CoilBit0071 := ContactBit0071;

// NETWORK 73
CoilBit0072 := ContactBit0072;

// NETWORK 74
CoilBit0073 := ContactBit0073;

// NETWORK 75
CoilBit0074 := ContactBit0074;

// NETWORK 76
CoilBit0075 := ContactBit0075;

// NETWORK 77
CoilBit0076 := ContactBit0076;

// NETWORK 78
CoilBit0077 := ContactBit0077;

// NETWORK 79
CoilBit0078 := ContactBit0078;

// NETWORK 80
CoilBit0079 := ContactBit0079;

// NETWORK 81
CoilBit0080 := ContactBit0080;

// NETWORK 82
CoilBit0081 := ContactBit0081;

// NETWORK 83
CoilBit0082 := ContactBit0082;

// NETWORK 84
CoilBit0083 := ContactBit0083;

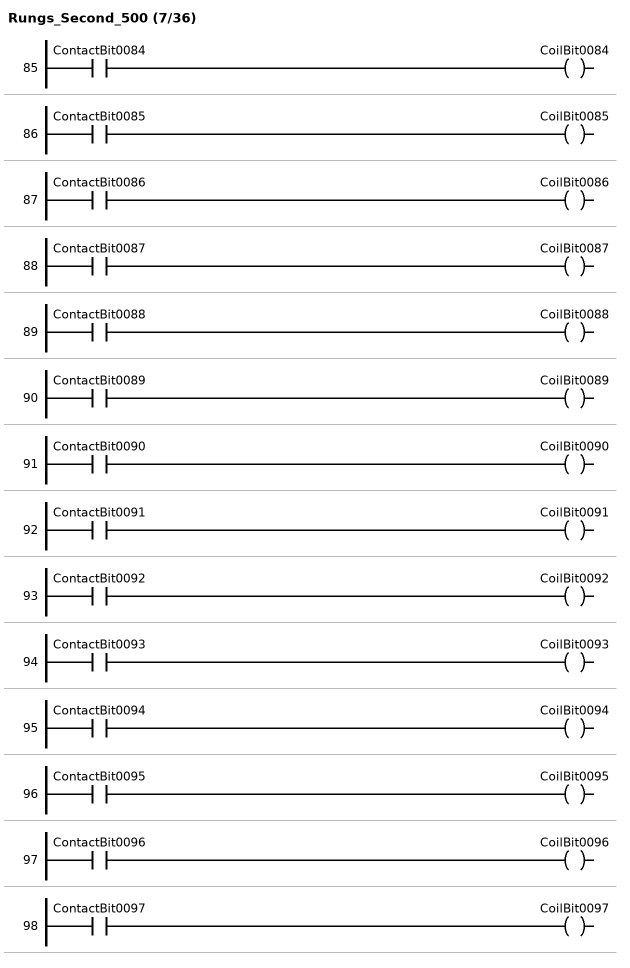
// NETWORK 85
CoilBit0084 := ContactBit0084;

// NETWORK 86
CoilBit0085 := ContactBit0085;

// NETWORK 87
CoilBit0086 := ContactBit0086;

// NETWORK 88
CoilBit0087 := ContactBit0087;

// NETWORK 89
CoilBit0088 := ContactBit0088;

// NETWORK 90
CoilBit0089 := ContactBit0089;

// NETWORK 91
CoilBit0090 := ContactBit0090;

// NETWORK 92
CoilBit0091 := ContactBit0091;

// NETWORK 93
CoilBit0092 := ContactBit0092;

// NETWORK 94
CoilBit0093 := ContactBit0093;

// NETWORK 95
CoilBit0094 := ContactBit0094;

// NETWORK 96
CoilBit0095 := ContactBit0095;

// NETWORK 97
CoilBit0096 := ContactBit0096;

// NETWORK 98
CoilBit0097 := ContactBit0097;

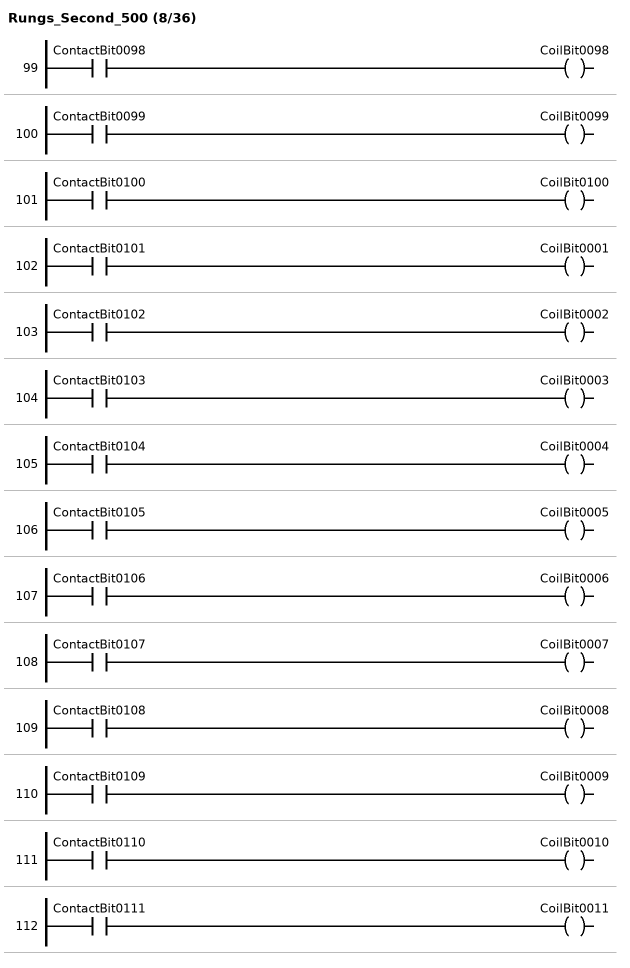
// NETWORK 99
CoilBit0098 := ContactBit0098;

// NETWORK 100
CoilBit0099 := ContactBit0099;

// NETWORK 101
CoilBit0100 := ContactBit0100;

// NETWORK 102
CoilBit0001 := ContactBit0101;

// NETWORK 103
CoilBit0002 := ContactBit0102;

// NETWORK 104
CoilBit0003 := ContactBit0103;

// NETWORK 105
CoilBit0004 := ContactBit0104;

// NETWORK 106
CoilBit0005 := ContactBit0105;

// NETWORK 107
CoilBit0006 := ContactBit0106;

// NETWORK 108
CoilBit0007 := ContactBit0107;

// NETWORK 109
CoilBit0008 := ContactBit0108;

// NETWORK 110
CoilBit0009 := ContactBit0109;

// NETWORK 111
CoilBit0010 := ContactBit0110;

// NETWORK 112
CoilBit0011 := ContactBit0111;

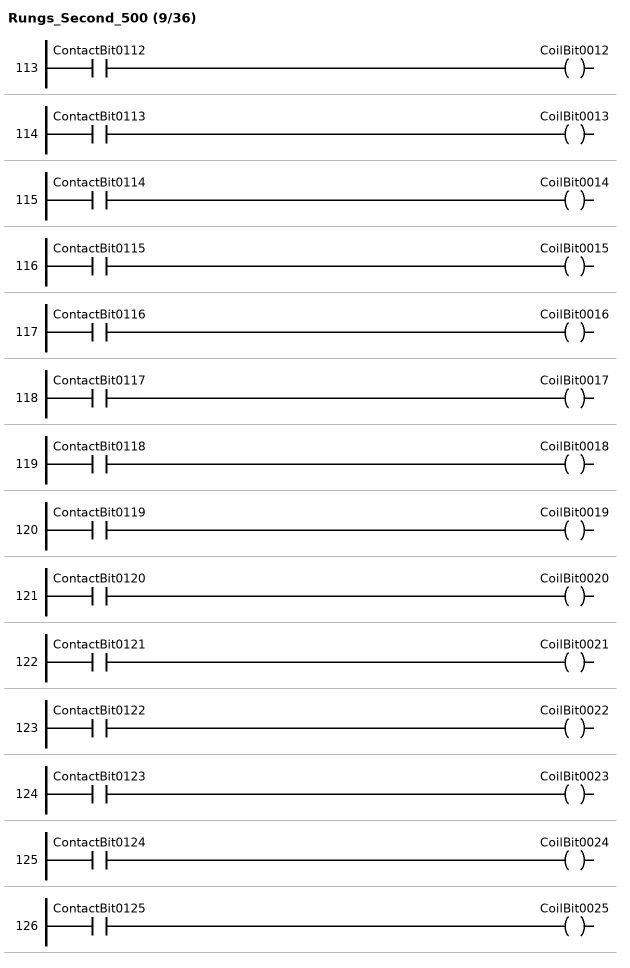
// NETWORK 113
CoilBit0012 := ContactBit0112;

// NETWORK 114
CoilBit0013 := ContactBit0113;

// NETWORK 115
CoilBit0014 := ContactBit0114;

// NETWORK 116
CoilBit0015 := ContactBit0115;

// NETWORK 117
CoilBit0016 := ContactBit0116;

// NETWORK 118
CoilBit0017 := ContactBit0117;

// NETWORK 119
CoilBit0018 := ContactBit0118;

// NETWORK 120
CoilBit0019 := ContactBit0119;

// NETWORK 121
CoilBit0020 := ContactBit0120;

// NETWORK 122
CoilBit0021 := ContactBit0121;

// NETWORK 123
CoilBit0022 := ContactBit0122;

// NETWORK 124
CoilBit0023 := ContactBit0123;

// NETWORK 125
CoilBit0024 := ContactBit0124;

// NETWORK 126
CoilBit0025 := ContactBit0125;

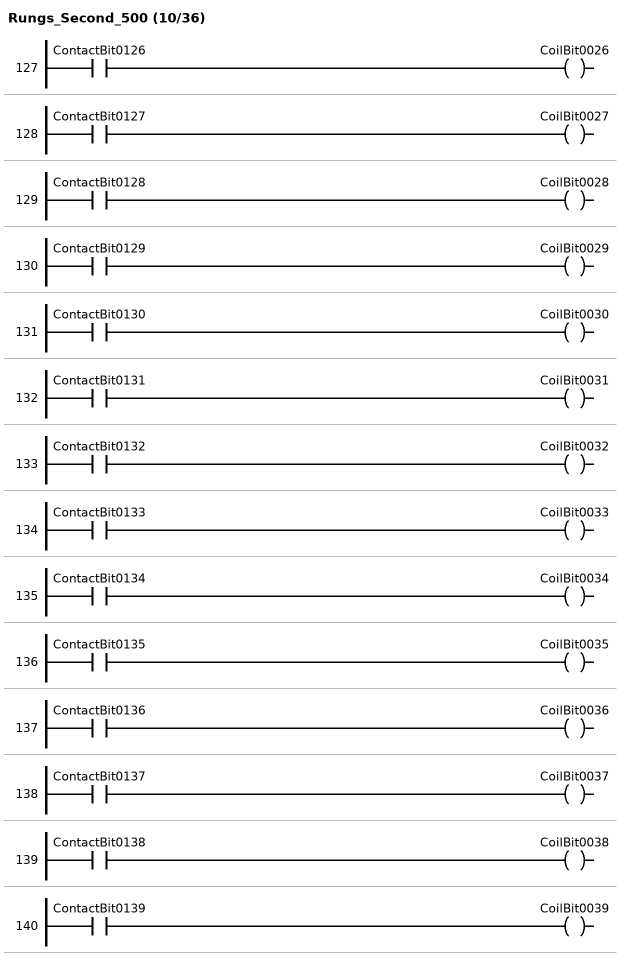
// NETWORK 127
CoilBit0026 := ContactBit0126;

// NETWORK 128
CoilBit0027 := ContactBit0127;

// NETWORK 129
CoilBit0028 := ContactBit0128;

// NETWORK 130
CoilBit0029 := ContactBit0129;

// NETWORK 131
CoilBit0030 := ContactBit0130;

// NETWORK 132
CoilBit0031 := ContactBit0131;

// NETWORK 133
CoilBit0032 := ContactBit0132;

// NETWORK 134
CoilBit0033 := ContactBit0133;

// NETWORK 135
CoilBit0034 := ContactBit0134;

// NETWORK 136
CoilBit0035 := ContactBit0135;

// NETWORK 137
CoilBit0036 := ContactBit0136;

// NETWORK 138
CoilBit0037 := ContactBit0137;

// NETWORK 139
CoilBit0038 := ContactBit0138;

// NETWORK 140
CoilBit0039 := ContactBit0139;

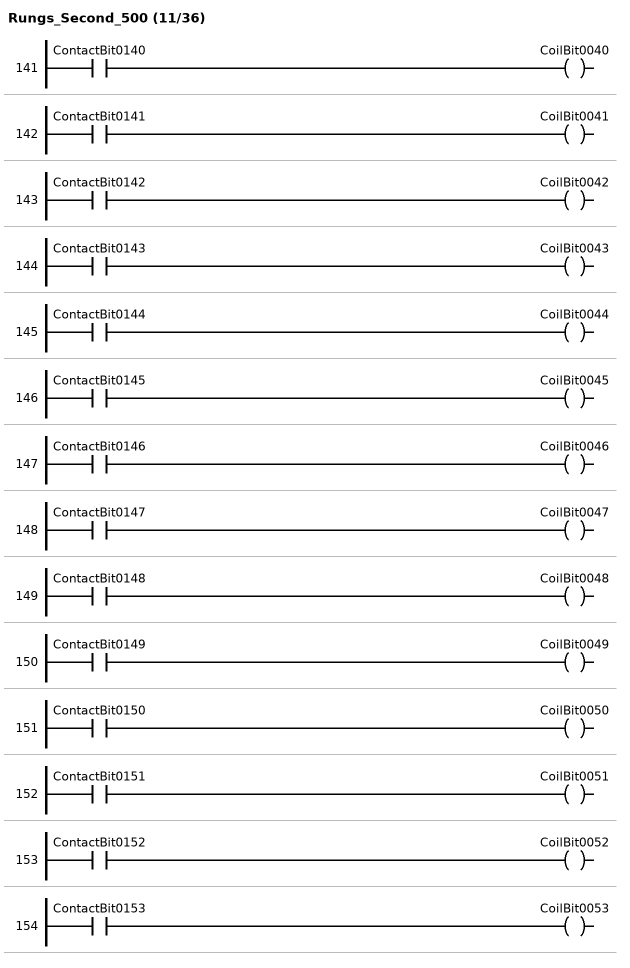
// NETWORK 141
CoilBit0040 := ContactBit0140;

// NETWORK 142
CoilBit0041 := ContactBit0141;

// NETWORK 143
CoilBit0042 := ContactBit0142;

// NETWORK 144
CoilBit0043 := ContactBit0143;

// NETWORK 145
CoilBit0044 := ContactBit0144;

// NETWORK 146
CoilBit0045 := ContactBit0145;

// NETWORK 147
CoilBit0046 := ContactBit0146;

// NETWORK 148
CoilBit0047 := ContactBit0147;

// NETWORK 149
CoilBit0048 := ContactBit0148;

// NETWORK 150
CoilBit0049 := ContactBit0149;

// NETWORK 151
CoilBit0050 := ContactBit0150;

// NETWORK 152
CoilBit0051 := ContactBit0151;

// NETWORK 153
CoilBit0052 := ContactBit0152;

// NETWORK 154
CoilBit0053 := ContactBit0153;

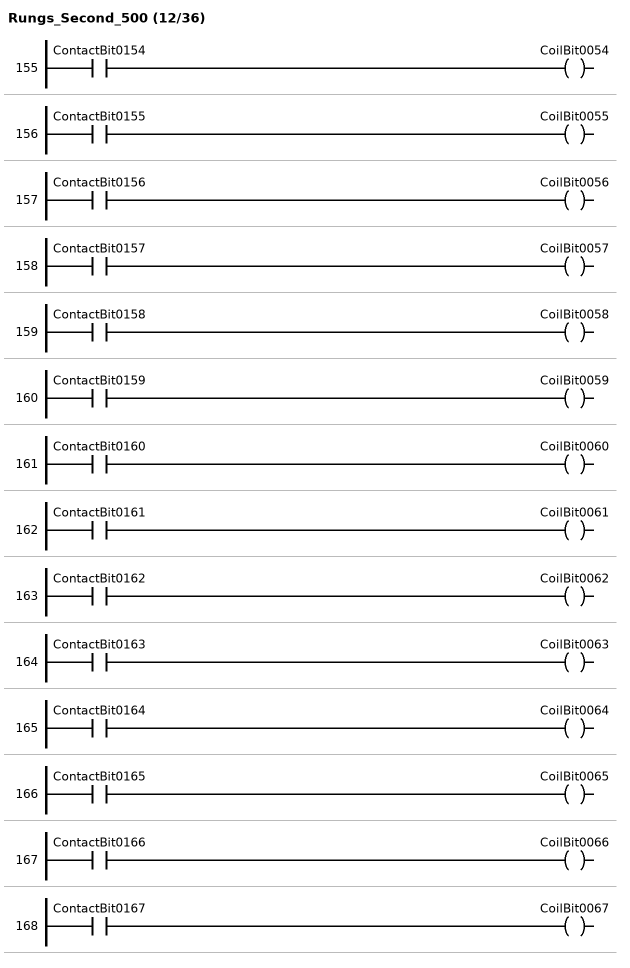
// NETWORK 155
CoilBit0054 := ContactBit0154;

// NETWORK 156
CoilBit0055 := ContactBit0155;

// NETWORK 157
CoilBit0056 := ContactBit0156;

// NETWORK 158
CoilBit0057 := ContactBit0157;

// NETWORK 159
CoilBit0058 := ContactBit0158;

// NETWORK 160
CoilBit0059 := ContactBit0159;

// NETWORK 161
CoilBit0060 := ContactBit0160;

// NETWORK 162
CoilBit0061 := ContactBit0161;

// NETWORK 163
CoilBit0062 := ContactBit0162;

// NETWORK 164
CoilBit0063 := ContactBit0163;

// NETWORK 165
CoilBit0064 := ContactBit0164;

// NETWORK 166
CoilBit0065 := ContactBit0165;

// NETWORK 167
CoilBit0066 := ContactBit0166;

// NETWORK 168
CoilBit0067 := ContactBit0167;

